// TIA Portal V17 export
// export: Created 2024-06-19T09:47:13.602572Z, ExportSetting WithDefaults, DisplayName Totally Integrated Automation Portal, DisplayVersion V17, DisplayName TIA Portal Openness, DisplayVersion V17, DisplayName TIA Portal Version Control Interface, DisplayVersion V17, DisplayName STEP 7 Professional, DisplayVersion V17, DisplayName STEP 7 Safety, DisplayVersion V17, DisplayName WinCC Professional, DisplayVersion V17
FUNCTION "G7A_St3" : Void   // FC310, LAD
{ S7_Optimized_Access := 'TRUE' }
VERSION : 0.1
// stored: AutoNumber false, IsIECCheckEnabled false, SetENOAutomatically false, UDAEnableTagReadback false
BEGIN

REGION Network 1: G7 Auto --> Station 3 : RX
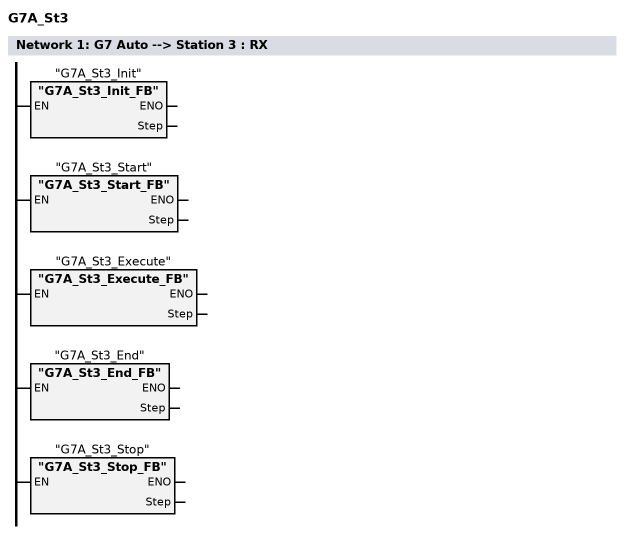
   RUNG wire#powerrail
      "G7A_St3_Init"("Step" =>)
   END_RUNG
   RUNG wire#powerrail
      "G7A_St3_Start"("Step" =>)
   END_RUNG
   RUNG wire#powerrail
      "G7A_St3_Execute"("Step" =>)
   END_RUNG
   RUNG wire#powerrail
      "G7A_St3_End"("Step" =>)
   END_RUNG
   RUNG wire#powerrail
      "G7A_St3_Stop"("Step" =>)
   END_RUNG
   // the same network as SCL:
   "G7A_St3_Init"();   // "G7A_St3_Init_FB"
   "G7A_St3_Start"();   // "G7A_St3_Start_FB"
   "G7A_St3_Execute"();   // "G7A_St3_Execute_FB"
   "G7A_St3_End"();   // "G7A_St3_End_FB"
   "G7A_St3_Stop"();   // "G7A_St3_Stop_FB"
END_REGION
END_FUNCTION
